Staubli VAL3: fileClose.pgx

program fileClose()
  local num l_nNum
begin
  for l_nNum=0 to 9
    $fileClose(l_nNum)
  endFor
end
